
FUNCTION CB_word_to_dword : DWORD

TITLE = ' Convert a word into a Double word '
VERSION : '1.0'
AUTHOR  : CB
NAME    : WorToDwo
FAMILY  : TNI

VAR_INPUT
    IN : WORD;
END_VAR

VAR_TEMP

END_VAR

BEGIN

CB_word_to_dword := WORD_TO_DWORD(IN);

END_FUNCTION
